// TwinCAT 3 PLC project PLC_CRIX_VAC
// Title: plc-crix-vac
// Company: SLAC - LCLS
// ProjectVersion: 0.0.0
// ProgramVersion: 3.1.4022.7
// libraries:
//   LCLS General, * (SLAC)
//   LCLS Sample Delivery, * (SLAC - LCLS)
//   LCLS Vacuum, * (SLAC - LCLS)
//   LCLSVacuumSerialDriverLib, * (SLAC - LCLS)
//   PMPS, * (SLAC - LCLS)
//   Tc2_SerialCom, * (Beckhoff Automation GmbH)
//   Tc2_Standard, * (Beckhoff Automation GmbH)
//   Tc2_System, * (Beckhoff Automation GmbH)
//   Tc3_Module, * (Beckhoff Automation GmbH)
// project tree:
//   / CommTask.TcTTO (not stored), PlcTask.TcTTO (not stored)
//   DUTs/ E_STATES.TcDUT (not stored)
//   GVLs/ GVL_ADS_Devices.TcGVL, GVL_Chamber_Gauges.TcGVL (not stored), GVL_Chamber_Valves.TcGVL (not stored), GVL_COM.TcGVL (not stored), GVL_COM_VLS.TcGVL (not stored), GVL_LI3K2.TcGVL (not stored), GVL_Mech_Room.TcGVL (not stored), GVL_PLC_Interfaces.TcGVL (not stored), GVL_PMPS.TcGVL (not stored), GVL_Pumps.TcGVL (not stored), GVL_Recirculation.TcGVL (not stored), GVL_Vars.TcGVL (not stored), GVL_VLS.TcGVL (not stored)
//   POUs/ FB_ChemRIXS_Turbo_ILK.TcPOU (not stored), F_TurboGateValve_Protection_ILK_Turbo_OFF_OK_NO_GPI_READ.TcPOU (not stored), MAIN.TcPOU (not stored), PRG_ADS_Gauges.TcPOU (not stored), PRG_ADS_Interfaces.TcPOU, PRG_Chamber_Gauges.TcPOU (not stored), PRG_Chamber_Pumps.TcPOU (not stored), PRG_Chamber_Valves.TcPOU (not stored), PRG_Com.TcPOU (not stored), PRG_COM_VLS.TcPOU (not stored), PRG_LI3K2.TcPOU (not stored), PRG_Mechanical_Room.TcPOU (not stored), PRG_MPS.TcPOU (not stored), PRG_RCC.TcPOU, PRG_VLS_Turbo.TcPOU (not stored), PRG_VLS_VACUUM.TcPOU (not stored), PRG_VLS_WINDOW.TcPOU (not stored)

// ---- GVLs/GVL_ADS_Devices.TcGVL
//{attribute 'qualified_only'}
VAR_GLOBAL

 {attribute 'pytmc' :=' pv: TM2K2:GCC:01:reader '}
    TM2K2_GCC_01_reader : FB_TGCC_ADS;
 {attribute 'pytmc' :=' pv: AT3K2:GCC:01:reader '}
    AT3K2_GCC_01_reader : FB_TGPI_ADS;

END_VAR

// ---- POUs/PRG_ADS_Interfaces.TcPOU
PROGRAM PRG_ADS_Interfaces
VAR

    // This variable needs to be instantiated for the Watchdog to work
    i_iWatchdog : UDINT;

    // create watch dog for LAMP PLC
    ads_watch_dog : FB_ADS_WATCHDOG;

END_VAR

TM2K2_GCC_01_reader(sNetId := '172.21.140.69.1.1', // AMS NET ID of RIXS vacuum PLC being read from
    nPort := 851, // ADS port of the PLC reading from this PLC
    sVarName := 'GVL_KFE_RIX_VAC.fb_TM2K2_K2B_GCC_1', // Full name of the FB containing the gauge to be read
    iWatchdog := i_iWatchdog // UDINT required for watchdog functionality
);

AT3K2_GCC_01_reader(sNetId := '172.21.140.69.1.1', // AMS NET ID of RIXS vacuum PLC being read from
    nPort := 851, // ADS port of the PLC reading from this PLC
    sVarName := 'GVL_KFE_RIX_VAC.fb_AT3K2_SOLID_GCP_1', // Full name of the FB containing the gauge to be read
    iWatchdog := i_iWatchdog // UDINT required for watchdog functionality
);

ads_watch_dog(
    sNetId := '172.21.140.69.1.1', // AMS NET ID of RIXS vacuum PLC reading from this PLC
    nPort := 851, // ADS port of the PLC reading from this PLC
    sVarName := 'GVL_RIX_INTF.ads_watch_dog', // the variable name of the watchdog on the remote plc
);

END_PROGRAM

// ---- POUs/PRG_RCC.TcPOU
PROGRAM PRG_RCC
VAR
    RCC_VRC_01_OPEN_OK : BOOL;
    RCC_VRC_02_OPEN_OK : BOOL;
    RCC_VRC_03_OPEN_OK : BOOL;
    RCC_VRC_04_OPEN_OK : BOOL;


    {attribute 'pytmc' :=' pv: CRIXS:RCC:GCP:01:ILK_Setpoint '}
    RCC_GCP_01_INTERLOCK_SETPOINT : REAL := 10;
	
	{attribute 'pytmc' :=' pv: CRIXS:RCC'}
	stRCC_CTL : ST_RCC;
	fbRCC 	  : FB_RCC;

END_VAR

RCC_GCP_01(PG=>);

RCC_STC_01();
RCC_STC_02();

fbRCC( stRCC_VRC_01:= RCC_VRC_01.iq_stValve,
	stRCC_VRC_02 := RCC_VRC_02.iq_stValve,
	stRCC_VRC_03 := RCC_VRC_03.iq_stValve,
	stRCC_VRC_04 := RCC_VRC_04.iq_stValve,
	stRCC_GCP_01 := RCC_GCP_01.PG,
	stRCC_CTL := stRCC_CTL
);

stRCC_CTL.xSystemOverrideMode_RCC := xSystemOverrideMode_RCC;
	


RCC_VRC_01(i_xExtILK_OK := stRCC_CTL.RCC_VRC_01_OPEN_OK,
                i_xOverrideMode := xSystemOverrideMode_RCC,
                 iq_stValve=> );

RCC_VRC_02(i_xExtILK_OK := stRCC_CTL.RCC_VRC_02_OPEN_OK,
                i_xOverrideMode := xSystemOverrideMode_RCC,
                 iq_stValve=> );


RCC_VRC_03(i_xExtILK_OK := stRCC_CTL.RCC_VRC_03_OPEN_OK,
                i_xOverrideMode := xSystemOverrideMode_RCC,
                 iq_stValve=> );


RCC_VRC_04(i_xExtILK_OK := stRCC_CTL.RCC_VRC_04_OPEN_OK,
                i_xOverrideMode := xSystemOverrideMode_RCC,
                 iq_stValve=> );

END_PROGRAM
